Fanuc KAREL source: ko00035.KL

PROGRAM KO00035
%STACKSIZE=65535
%PRIORITY=65535
%NOLOCKGROUP
VAR
P1 : POSITION
P2 : POSITION
F : BOOLEAN
OUT : XYZWPREXT
BEGIN
F=TRUE
-- UNSAFE_SOURCE_IR line 11: OUT = MIRROR(convert_position_to_xyzwprext(P1), P2, F)
END KO00035
